{attribute 'qualified_only'}
{attribute 'strict'}
{attribute 'to_string'}
TYPE eSystemCommand :
(
	KEINE		:= 0,
	AUSCHALTEN 	:= 1,
	EINSCHALTEN := 2,
	STOPPEN		:= 3,
	RESETTEN	:= 4
);
END_TYPE

(* stored: Version 1.1.0.1
   DUT eSystemCommand: Id {92e17196-33c3-4aa3-a08b-5908cd2d45b5} *)
